// Brief: Slave Arm test
FUNCTION_BLOCK PUBLIC FB_SlaveCtrlInstruAutoTest_bak EXTENDS FB_SlaveArmCtrlBase
VAR CONSTANT
	m_instruOpenGripMoveTrajNum :INT :=18;
	m_instruGripMoveTrajNum :INT :=8;
	m_instruYawRange :LREAL := 75 * g_deg2Rad;
END_VAR
VAR
	// test mode. 
	//0: auto test - finger grip and release
	//1: auto test - finger open and mvoe
	//2: auto test - finger grip and move
	m_instruTestMode :INT := 0;
	m_lastInstruTestMode :INT := 0;
	
	// variables for auto test
	m_autoTestCycles :INT :=0;
	m_autoTestStep :INT :=0;

	// final target DH joint position and grip angle
	m_targetDHJntPos:Vec3d;
	m_targetGripAng:LREAL;
	m_targetGripForceLevel :LREAL :=0;
	
	// interploated command joint position and grip angle 
	m_cmdDHJntPos :Vec6d;
	m_cmdDHJntVel :Vec6d;
	m_cmdGripAng:LREAL;

	// last joint position 
	m_lastCmdJntPos :Vec8d ;
	
	// instrument controller
	m_instruController : FB_BasicInstruControl;
	m_usKnifeController : FB_UltrosonicKnifeControl;
	m_instruCmdJntPos,m_instruCmdJntVel : Vec5d;
	m_instruCmdJntTrq :Vec5d;
	
	// OTG
	m_DHJntOTG:ARRAY[1..3] OF FB_secOrdTrajFilter;
	m_gripAngleOTG : FB_secOrdTrajFilter;
	m_maxJntVel:Vec3d:=[3(2.0)];
	m_maxJntAcc:Vec3d:=[3(4.0)];
	
	// instrument open and grip move motion via points[roll, pitch, yaw]
	m_openGripStep :INT :=0;
	m_gripOpenStep :INT :=0;
	m_instruOpenGrioMovePos:ARRAY [1..m_instruOpenGripMoveTrajNum, 1..3] OF LREAL:=
	// move with gripper close
	[0,		-pi/2,		0,	
	0,		-pi/2,		pi/3,	
	0,		-pi/2,		-pi/3,
	0,		-pi/2+m_instruYawRange,		0,
	0,		-pi/2+m_instruYawRange,		pi/3,
	0,		-pi/2+m_instruYawRange,		-pi/3,
	0,		-pi/2-m_instruYawRange,		0,
	0,		-pi/2-m_instruYawRange,		-pi/3,
	0,		-pi/2-m_instruYawRange,		pi/3,
	// move with gripper open
	pi,		-pi/2,		0,	
	pi,		-pi/2,		pi/3,	
	pi,		-pi/2,		-pi/3,
	pi,		-pi/2+m_instruYawRange,		0,
	pi,		-pi/2+m_instruYawRange,		pi/3,
	pi,		-pi/2+m_instruYawRange,		-pi/3,
	pi,		-pi/2-m_instruYawRange,		0,
	pi,		-pi/2-m_instruYawRange,		-pi/3,
	pi,		-pi/2-m_instruYawRange,		pi/3];
	
	// instrument move motion via points[roll, pitch, yaw]
	m_instruGripMovePos:ARRAY [1..m_instruGripMoveTrajNum, 1..3] OF LREAL:=
	// move with gripper close
	[0,		-pi/2+m_instruYawRange,		pi/3,
	0,		-pi/2+m_instruYawRange,		-pi/3,
	0,		-pi/2-m_instruYawRange,		pi/3,
	0,		-pi/2-m_instruYawRange,		-pi/3,
	pi,		-pi/2+m_instruYawRange,		pi/3,
	pi,		-pi/2+m_instruYawRange,		-pi/3,
	pi,		-pi/2-m_instruYawRange,		pi/3,
	pi,		-pi/2-m_instruYawRange,		-pi/3];
	
	// instrument tyep
	m_instruType : E_InstrumentType;
																				
END_VAR

METHOD PROTECTED calcCmdJntPos : BOOL
VAR_IN_OUT CONSTANT
	i_endoscopePose : ST_Frame;
	i_masterStatus :ST_MasterStatus;
	i_setupStatus: ST_SetupStatus;
	i_slaveArm :FB_SlaveArm;
END_VAR

VAR 
	i:INT :=0;
	errThres :LREAL;

END_VAR

IF GVL_InstruTestUIVars.g_maxInstruAutoTestCycles > 0 AND m_autoTestCycles > GVL_InstruTestUIVars.g_maxInstruAutoTestCycles THEN
	RETURN;
END_IF

// determine final target DH joint position
CASE m_instruTestMode OF
	0:
		fingerOpenCloseTest(i_slaveArm);
	1:
		fingerOpenGripMoveTest(i_slaveArm);
	2:
		fingerGripMoveTest(i_slaveArm);
	ELSE
		RETURN;
END_CASE

// run OTG
FOR i:=1 TO 3  DO
	m_DHJntOTG[i].run(m_targetDHJntPos[i],0.0, o_cmdAcc=>,o_cmdVel=>m_cmdDHJntVel[i],o_cmdPos=> m_cmdDHJntPos[i+3]);
END_FOR
m_gripAngleOTG.run(m_targetGripAng,0.0, o_cmdAcc=>,o_cmdVel=>,o_cmdPos=>m_cmdGripAng);

// calculate target motor joint position from DH joint position
i_slaveArm.instrument.instruIK(m_cmdDHJntPos,m_cmdGripAng, o_jntPos=>m_cmdJntPos);

// command velocity
vecSub(m_cmdJntPos, m_lastCmdJntPos, m_cmdJntVel);
vecSelfMultiNum(m_cmdJntVel, g_slaveArmCtrlFreq);
m_lastCmdJntPos:=m_cmdJntPos;

m_lastInstruTestMode := m_instruTestMode;
END_METHOD

// override this function in each exact controller
METHOD PROTECTED calcCmdJntTrq : BOOL
VAR_IN_OUT CONSTANT
	i_endoscopePose : ST_Frame;
	i_masterStatus :ST_MasterStatus;
	i_setupStatus: ST_SetupStatus;
	i_slaveArm :FB_SlaveArm;
END_VAR

VAR 
	nullspaceMat :Mat7d;
	ctrlTrq : Vec7d;
	i : int ;
END_VAR
// set joint torque to zero in default
m_cmdJntTrq := g_zeroVec8d;

// instrument joint control
FOR i:=1 TO 5 DO 
	m_instruCmdJntPos[i]:=m_cmdJntPos[i+3];
	m_instruCmdJntVel[i]:=m_cmdJntVel[i+3];
END_FOR

IF i_slaveArm.instrument.instruType = InstruType_UltrasoundKnifeS OR i_slaveArm.instrument.instruType = InstruType_UltrasoundKnifeU THEN
	m_usKnifeController.run(m_instruCmdJntPos,m_instruCmdJntVel, m_targetGripForceLevel, i_slaveArm, o_cmdJntTrq=>m_instruCmdJntTrq);
ELSE
	m_instruController.run(m_instruCmdJntPos,m_instruCmdJntVel, m_cmdDHJntPos[6], m_cmdDHJntVel[6], m_targetGripForceLevel, i_slaveArm, o_cmdJntTrq=>m_instruCmdJntTrq);
END_IF

FOR i:=1 TO 5 DO
	m_cmdJntTrq[i+3]:=m_instruCmdJntTrq[i];
END_FOR
END_METHOD

METHOD fingerGripMoveTest : BOOL
VAR_IN_OUT CONSTANT
	i_slaveArm :FB_SlaveArm;
END_VAR
VAR
	i:INT;
END_VAR

m_targetGripForceLevel :=100;
m_autoTestStep := LIMIT(0,m_autoTestStep, m_instruGripMoveTrajNum-1);
FOR i:=1 TO 3 DO
	 m_targetDHJntPos[i] := m_instruGripMovePos[m_autoTestStep+1, i];
END_FOR
	 
IF ABS(m_cmdDHJntPos[4]-m_targetDHJntPos[1])< g_jntCtrlAngTolLow AND ABS(m_cmdDHJntPos[5]-m_targetDHJntPos[2])< g_jntCtrlAngTolLow 
		AND ABS(m_cmdDHJntPos[6]-m_targetDHJntPos[3])< g_jntCtrlAngTolLow  THEN
	m_autoTestStep :=m_autoTestStep + 1;
END_IF
 
IF m_autoTestStep >= m_instruGripMoveTrajNum THEN
	m_autoTestCycles := m_autoTestCycles + 1;
	m_autoTestStep := 0;
END_IF
END_METHOD

METHOD fingerGripOpenOnce : BOOL
VAR_IN_OUT CONSTANT
	i_slaveArm :FB_SlaveArm;
END_VAR
CASE m_gripOpenStep OF
	0:
		m_targetGripAng := 0;
		m_targetGripForceLevel :=0;
	1:
		m_targetGripAng := g_minSlaveGripAngle;
		m_targetGripForceLevel :=0;		
	2:
		m_targetGripAng := -45* g_deg2rad;
		m_targetGripForceLevel :=100;
	3:
		m_targetGripAng := g_minSlaveGripAngle;
		m_targetGripForceLevel :=100;

	4:
		m_targetGripAng := g_minSlaveGripAngle;
		m_targetGripForceLevel :=0;
END_CASE

IF ABS(m_cmdGripAng- m_targetGripAng)< g_jntCtrlAngTolLow THEN
	 m_gripOpenStep :=m_gripOpenStep + 1;
END_IF

fingerGripOpenOnce := m_gripOpenStep > 4;
END_METHOD

METHOD fingerOpenCloseTest : BOOL
VAR_IN_OUT CONSTANT
	i_slaveArm :FB_SlaveArm;
END_VAR
m_autoTestStep := LIMIT(0,m_autoTestStep, 5);
CASE m_autoTestStep OF
	0:
		m_targetGripAng := 0;
		m_targetGripForceLevel :=0;
	1:
		m_targetGripAng := GVL_InstruTestUIVars.g_maxGripAng * g_deg2Rad;//i_slaveArm.instrument.instruTypeInfo.m_maxGripAngle;
		m_targetGripForceLevel :=0;
	2:
		m_targetGripAng := g_minSlaveGripAngle;
		m_targetGripForceLevel :=0;
	3:
		m_targetGripAng := -pi/2;
		m_targetGripForceLevel :=100;
	4:
		m_targetGripAng := g_minSlaveGripAngle;
		m_targetGripForceLevel :=100;
	5:
		m_targetGripAng := 0;
		m_targetGripForceLevel :=0;
END_CASE

IF ABS(m_cmdGripAng- m_targetGripAng)< g_jntCtrlAngTolLow THEN
	 m_autoTestStep :=m_autoTestStep + 1;
END_IF

IF m_autoTestStep > 5 THEN
	m_autoTestCycles := m_autoTestCycles + 1;
	m_autoTestStep := 0;
END_IF
END_METHOD

METHOD fingerOpenGripMoveTest : BOOL
VAR_IN_OUT CONSTANT
	i_slaveArm :FB_SlaveArm;
END_VAR
VAR
	i:INT;
	fingerMotionFlag : BOOL;
END_VAR
m_autoTestStep := LIMIT(0,m_autoTestStep, m_instruOpenGripMoveTrajNum-1);
FOR i:=1 TO 3 DO
	 m_targetDHJntPos[i] := m_instruOpenGrioMovePos[m_autoTestStep+1, i];
END_FOR
	 
IF ABS(m_cmdDHJntPos[4]-m_targetDHJntPos[1])< g_jntCtrlAngTolLow AND ABS(m_cmdDHJntPos[5]-m_targetDHJntPos[2])< g_jntCtrlAngTolLow 
		AND ABS(m_cmdDHJntPos[6]-m_targetDHJntPos[3])< g_jntCtrlAngTolLow  THEN
	
	IF m_autoTestStep < m_instruOpenGripMoveTrajNum/2 THEN
		fingerMotionFlag:=fingerOpenGripOnce(i_slaveArm);
	ELSE
		fingerMotionFlag:=fingerGripOpenOnce(i_slaveArm);
	END_IF
	
	IF fingerMotionFlag THEN
		m_autoTestStep :=m_autoTestStep + 1;
		m_openGripStep :=0;
		m_gripOpenStep :=0;
	END_IF
	
END_IF
 
IF m_autoTestStep >= m_instruOpenGripMoveTrajNum THEN
	m_autoTestCycles := m_autoTestCycles + 1;
	m_autoTestStep := 0;
END_IF
END_METHOD

METHOD fingerOpenGripOnce : BOOL
VAR_IN_OUT CONSTANT
	i_slaveArm :FB_SlaveArm;
END_VAR
CASE m_openGripStep OF
	0:
		m_targetGripAng := 0;
		m_targetGripForceLevel :=0;
	1:
		m_targetGripAng := GVL_InstruTestUIVars.g_maxGripAng * g_deg2Rad;//i_slaveArm.instrument.instruTypeInfo.m_maxGripAngle;
		m_targetGripForceLevel :=0;
	2:
		m_targetGripAng := g_minSlaveGripAngle;
		m_targetGripForceLevel :=0;
	3:
		m_targetGripAng := -45 * g_deg2rad;
		m_targetGripForceLevel :=100;
	4:
		m_targetGripAng := g_minSlaveGripAngle;
		m_targetGripForceLevel :=100;
END_CASE

IF ABS(m_cmdGripAng- m_targetGripAng)< g_jntCtrlAngTolLow THEN
	 m_openGripStep :=m_openGripStep + 1;
END_IF

fingerOpenGripOnce := m_openGripStep > 4;
END_METHOD

METHOD PUBLIC init : BOOL
VAR_IN_OUT CONSTANT
	i_slaveArm	:FB_SlaveArm;
END_VAR
VAR_IN_OUT 
	r_slaveArmCtrlCmd :ST_SlaveArmCtrlCmds;
END_VAR

VAR
	i:int;
END_VAR
SUPER^.Init(i_slaveArm,r_slaveArmCtrlCmd);
m_lastCmdJntPos:=m_cmdJntPos;
m_jntOPMode[1] := DriverOPMode_PosTrq;
m_jntOPMode[2] := DriverOPMode_PosTrq;
m_jntOPMode[3] := DriverOPMode_PosTrq;
m_jntOPMode[4] := DriverOPMode_Trq;
m_jntOPMode[5] := DriverOPMode_Trq;
m_jntOPMode[6] := DriverOPMode_Trq;
m_jntOPMode[7] := DriverOPMode_Trq;
m_jntOPMode[8] := DriverOPMode_Trq;

m_instruTestMode := GVL_InstruTestUIVars.g_instruAutoTestMode;
m_autoTestStep:=0 ;
m_autoTestCycles := 0;
m_openGripStep :=0;
m_gripOpenStep :=0;
m_cmdDHJntPos :=i_slaveArm.curDHJntPos;
m_cmdDHJntVel :=g_zeroVec6d;
m_targetGripAng := i_slaveArm.curGripAngle;
m_targetDHJntPos[1] := i_slaveArm.curDHJntPos[4];
m_targetDHJntPos[2] := i_slaveArm.curDHJntPos[5];
m_targetDHJntPos[3] := i_slaveArm.curDHJntPos[6];

// init instrument controller
m_instruController.init(i_slaveArm);
m_usKnifeController.init(i_slaveArm);
m_instruType := i_slaveArm.instrument.instruType;

FOR i:=1 TO 3  DO
	m_DHJntOTG[i].init(m_cmdDHJntPos[i+3], 0, m_maxJntVel[i], m_maxJntAcc[i], g_slaveArmCtrlCycleTime);
END_FOR

m_gripAngleOTG.init(m_targetGripAng, 0, m_maxJntVel[3], m_maxJntAcc[3], g_slaveArmCtrlCycleTime);
// update commands to arm
copyCmds(r_slaveArmCtrlCmd);
END_METHOD

PROPERTY InstruBacklash : Vec5d
GET
IF m_instruType = InstruType_UltrasoundKnifeS OR m_instruType = InstruType_UltrasoundKnifeU THEN
	instruBacklash := g_zeroVec5d;
ELSE
	instruBacklash := m_instruController.m_jntBacklash;
END_IF
END_GET
END_PROPERTY

END_FUNCTION_BLOCK

(* stored: Version 1.1.0.1, ProductVersion 3.1.4024.12
   POU FB_SlaveCtrlInstruAutoTest_bak: Id {d70115e7-7668-49fd-9f57-bdf3458ba446}, SpecialFunc None
   Method calcCmdJntPos: Id {fabdb455-5225-4307-a367-b36816d27b6f}
   Method calcCmdJntTrq: Id {89cc8590-b0ea-4a29-944b-9b994680a8df}
   Method fingerGripMoveTest: Id {b23b170a-3eed-478e-a97c-17d1ca24b714}
   Method fingerGripOpenOnce: Id {eecdcd4b-6163-4fb0-ac83-a217b04d8eb3}
   Method fingerOpenCloseTest: Id {7cc8daed-3bf9-42ca-9d17-f827b074e621}
   Method fingerOpenGripMoveTest: Id {9c6e0ab8-ec0f-4e57-8c89-55d8aad6317c}
   Method fingerOpenGripOnce: Id {b00fafe9-f130-44f7-ad16-8ec8acf445cf}
   Method init: Id {1224d61d-417a-4654-acf9-99ef0220f449}
   Property InstruBacklash: Id {36c2eae9-d34a-4d78-a1ca-ae4b84eb11b6}
   Get Get: Id {a50be6d4-ea37-4d42-9226-d0fdbcd75516} *)
